FUNCTION_BLOCK TestPublishValue
  VAR
    MQTT : HANDLE_MQTT;
    MQTT_INFO : MQTT_INFO;
    MQTT_IN_OUT : MQTT_IN_OUT;
    testPiublish : ARRAY[0..100] OF MQTTPublish;  (* testPiublish: SD_MQTT.MQTTPublish; *)
    init : BOOL := FALSE;
    sendTest : BOOL;
    TestValue : ARRAY[0..99] OF MQTTValue;
    testtime : ton;
    i : UDINT;
    qos : QoS := 2;
    sub1 : MQTTSubscribe;
    Values : ARRAY[0..99] OF CommonTypesAndFunctions.ALL_TYPES_UNION;
    temp1 : LREAL;
    tmpPointer : CommonTypesAndFunctions.ALL_TYPES_UNION_POINTER;
    MQTTretain : BOOL := TRUE;
    enable : BOOL;
    ERROR_C : DWORD;
    ERROR_T : BYTE;
    ValueTime : TIME := TIME#5s0ms;
  END_VAR

            MQTT_IN_OUT.ClientID :='testCodesys';
MQTT_IN_OUT.COM_CONFIG.MaxPayloadSize :=50000;
MQTT_IN_OUT.COM_CONFIG.MaxTopicLevels := 200;
//testtime(IN:= , PT:= );
testtime(IN:= NOT testtime.Q AND sendTest, PT:= T#100MS);

//testtime(IN:= NOT testtime.Q AND sendTest, PT:= T#10S);
IF NOT init THEN
	init := TRUE;
	tmpPointer.POINTER_TO_LREAL_T := ADR(temp1);
	TestValue[0].Init(
	Topic:= ADR('Haus/Raum1/Tisch/'), 
	ValueName:= ADR('Temperatur'), 
	ValuePointer:= tmpPointer, 
	ValueType:= CommonTypesAndFunctions.VAR_TYPES.LREAL_T, 
	ValueDiff:= 1, 
	MQTT_IN_OUT:= ADR(MQTT_IN_OUT), 
	DecimalPlace:= 2, 
	QoS:= qos, 
	RetainMqtt:= MQTTretain,
	MinTime:=ValueTime);
	sub1.SetMqttInOut(MQTT_IN_OUT:= ADR(MQTT_IN_OUT));

END_IF
TestValue[0]();


MQTT(
	MQTT_INFO:= MQTT_INFO, 
	MQTT_IN_OUT:= MQTT_IN_OUT, 
	ENABLE:= enable, 
	URL:= 'windows-10-pro:1883', 
	TIMEOUT:= T#5S, 
	ERROR_C=> ERROR_C, 
	ERROR_T=> ERROR_T);
          
END_FUNCTION_BLOCK

FUNCTION_BLOCK TestSubscribeOld
  VAR
    MQTT_IN_OUT : MQTT_IN_OUT;
    subscribe : ARRAY[0..20] OF MQTTSubscribe;
    init : BOOL;
    i : INT;
    recived : ARRAY[0..20] OF BOOL;
    CountSplitTopicSizeExceeded : ULINT;
  END_VAR

            IF NOT init THEN
	init := TRUE;
	FOR i := 0 TO 20 DO
		subscribe[i].SetMqttInOut(MQTT_IN_OUT:= ADR(MQTT_IN_OUT));
	END_FOR
END_IF
//MQTT_IN_OUT.OUT.DataRecived := TRUE;
MQTT_IN_OUT.InFree := TRUE;
(*
MQTT_IN_OUT.OUT.MqttTopic := 'r//test';
//GetSplitTopic(in:= MQTT_IN_OUT.OUT.MqttTopic, Target:= ADR(MQTT_IN_OUT.OUT.Topics), CountSplitTopicSizeExceeded:= ADR(CountSplitTopicSizeExceeded));
i:=0;
subscribe[i](
	Subscribe:= TRUE, 
	Topic:= '+//test', 
	QoSSubscribe:= 0, 
	Payload=> , 
	TopicOut=> , 
	SendTimeout=> , 
	SubscribeFail=> , 
	TopicValid=> , 
	Recived=> recived[i]);
MQTT_IN_OUT.OUT.MqttTopic := '/rest/zt';
//GetSplitTopic(in:= MQTT_IN_OUT.OUT.MqttTopic, Target:= ADR(MQTT_IN_OUT.OUT.Topics), CountSplitTopicSizeExceeded:= ADR(CountSplitTopicSizeExceeded));
i:=i+1;
subscribe[i](
	Subscribe:= TRUE, 
	Topic:= '#', 
	QoSSubscribe:= 0, 
	Payload=> , 
	TopicOut=> , 
	SendTimeout=> , 
	SubscribeFail=> , 
	TopicValid=> , 
	Recived=> recived[i]);
MQTT_IN_OUT.OUT.MqttTopic := '566//test/3565/356';
//GetSplitTopic(in:= MQTT_IN_OUT.OUT.MqttTopic, Target:= ADR(MQTT_IN_OUT.OUT.Topics), CountSplitTopicSizeExceeded:= ADR(CountSplitTopicSizeExceeded));
i:=i+1;
subscribe[i](
	Subscribe:= TRUE, 
	Topic:= '+//test/#', 
	QoSSubscribe:= 0, 
	Payload=> , 
	TopicOut=> , 
	SendTimeout=> , 
	SubscribeFail=> , 
	TopicValid=> , 
	Recived=> recived[i]);
MQTT_IN_OUT.OUT.MqttTopic := 'test';
//GetSplitTopic(in:= MQTT_IN_OUT.OUT.MqttTopic, Target:= ADR(MQTT_IN_OUT.OUT.Topics), CountSplitTopicSizeExceeded:= ADR(CountSplitTopicSizeExceeded));
i:=i+1;
subscribe[i](
	Subscribe:= TRUE, 
	Topic:= 'test', 
	QoSSubscribe:= 0, 
	Payload=> , 
	TopicOut=> , 
	SendTimeout=> , 
	SubscribeFail=> , 
	TopicValid=> , 
	Recived=> recived[i]);
MQTT_IN_OUT.OUT.MqttTopic := '/test/';
//GetSplitTopic(in:= MQTT_IN_OUT.OUT.MqttTopic, Target:= ADR(MQTT_IN_OUT.OUT.Topics), CountSplitTopicSizeExceeded:= ADR(CountSplitTopicSizeExceeded));
i:=i+1;
subscribe[i](
	Subscribe:= TRUE, 
	Topic:= 'test/', 
	QoSSubscribe:= 0, 
	Payload=> , 
	TopicOut=> , 
	SendTimeout=> , 
	SubscribeFail=> , 
	TopicValid=> , 
	Recived=> recived[i]);
MQTT_IN_OUT.OUT.MqttTopic := 'test/test1';
//GetSplitTopic(in:= MQTT_IN_OUT.OUT.MqttTopic, Target:= ADR(MQTT_IN_OUT.OUT.Topics), CountSplitTopicSizeExceeded:= ADR(CountSplitTopicSizeExceeded));
i:=i+1;
subscribe[i](
	Subscribe:= TRUE, 
	Topic:= 'test/test1', 
	QoSSubscribe:= 0, 
	Payload=> , 
	TopicOut=> , 
	SendTimeout=> , 
	SubscribeFail=> , 
	TopicValid=> , 
	Recived=> recived[i]);
MQTT_IN_OUT.OUT.MqttTopic := 'a/ret/test';
//GetSplitTopic(in:= MQTT_IN_OUT.OUT.MqttTopic, Target:= ADR(MQTT_IN_OUT.OUT.Topics), CountSplitTopicSizeExceeded:= ADR(CountSplitTopicSizeExceeded));
i:=i+1;
subscribe[i](
	Subscribe:= TRUE, 
	Topic:= 'a/+/test', 
	QoSSubscribe:= 0, 
	Payload=> , 
	TopicOut=> , 
	SendTimeout=> , 
	SubscribeFail=> , 
	TopicValid=> , 
	Recived=> recived[i]);
MQTT_IN_OUT.OUT.MqttTopic := '/test/etwetre/';
//GetSplitTopic(in:= MQTT_IN_OUT.OUT.MqttTopic, Target:= ADR(MQTT_IN_OUT.OUT.Topics), CountSplitTopicSizeExceeded:= ADR(CountSplitTopicSizeExceeded));
i:=i+1;
subscribe[i](
	Subscribe:= TRUE, 
	Topic:= '/test/+',//no match !!!!!
	QoSSubscribe:= 0, 
	Payload=> , 
	TopicOut=> , 
	SendTimeout=> , 
	SubscribeFail=> , 
	TopicValid=> , 
	Recived=> recived[i]);
MQTT_IN_OUT.OUT.MqttTopic := '/test/etwetre';
//GetSplitTopic(in:= MQTT_IN_OUT.OUT.MqttTopic, Target:= ADR(MQTT_IN_OUT.OUT.Topics), CountSplitTopicSizeExceeded:= ADR(CountSplitTopicSizeExceeded));
i:=i+1;
subscribe[i](
	Subscribe:= TRUE, 
	Topic:= '/test/+',//match !!!!!!
	QoSSubscribe:= 0, 
	Payload=> , 
	TopicOut=> , 
	SendTimeout=> , 
	SubscribeFail=> , 
	TopicValid=> , 
	Recived=> recived[i]);
MQTT_IN_OUT.OUT.MqttTopic := '/finance';
//GetSplitTopic(in:= MQTT_IN_OUT.OUT.MqttTopic, Target:= ADR(MQTT_IN_OUT.OUT.Topics), CountSplitTopicSizeExceeded:= ADR(CountSplitTopicSizeExceeded));
i:=i+1;
subscribe[i](
	Subscribe:= TRUE, 
	Topic:= '+/+', //match
	QoSSubscribe:= 0, 
	Payload=> , 
	TopicOut=> , 
	SendTimeout=> , 
	SubscribeFail=> , 
	TopicValid=> , 
	Recived=> recived[i]);
MQTT_IN_OUT.OUT.MqttTopic := '/finance';
//GetSplitTopic(in:= MQTT_IN_OUT.OUT.MqttTopic, Target:= ADR(MQTT_IN_OUT.OUT.Topics), CountSplitTopicSizeExceeded:= ADR(CountSplitTopicSizeExceeded));
i:=i+1;
subscribe[i](
	Subscribe:= TRUE, 
	Topic:= '/+', //match
	QoSSubscribe:= 0, 
	Payload=> , 
	TopicOut=> , 
	SendTimeout=> , 
	SubscribeFail=> , 
	TopicValid=> , 
	Recived=> recived[i]);
MQTT_IN_OUT.OUT.MqttTopic := '/finance';
//GetSplitTopic(in:= MQTT_IN_OUT.OUT.MqttTopic, Target:= ADR(MQTT_IN_OUT.OUT.Topics), CountSplitTopicSizeExceeded:= ADR(CountSplitTopicSizeExceeded));
i:=i+1;
subscribe[i](
	Subscribe:= TRUE, 
	Topic:= '+',//no match 
	QoSSubscribe:= 0, 
	Payload=> , 
	TopicOut=> , 
	SendTimeout=> , 
	SubscribeFail=> , 
	TopicValid=> , 
	Recived=> recived[i]);
MQTT_IN_OUT.OUT.MqttTopic := 'finance/test';
//GetSplitTopic(in:= MQTT_IN_OUT.OUT.MqttTopic, Target:= ADR(MQTT_IN_OUT.OUT.Topics), CountSplitTopicSizeExceeded:= ADR(CountSplitTopicSizeExceeded));
i:=i+1;
subscribe[i](
	Subscribe:= TRUE, 
	Topic:= 'finance/test/',//** 
	QoSSubscribe:= 0, 
	Payload=> , 
	TopicOut=> , 
	SendTimeout=> , 
	SubscribeFail=> , 
	TopicValid=> , 
	Recived=> recived[i]);
MQTT_IN_OUT.OUT.MqttTopic := 'finance/test';
//GetSplitTopic(in:= MQTT_IN_OUT.OUT.MqttTopic, Target:= ADR(MQTT_IN_OUT.OUT.Topics), CountSplitTopicSizeExceeded:= ADR(CountSplitTopicSizeExceeded));
i:=i+1;
subscribe[i](
	Subscribe:= TRUE, 
	Topic:= 'finance/test',//?? 
	QoSSubscribe:= 0, 
	Payload=> , 
	TopicOut=> , 
	SendTimeout=> , 
	SubscribeFail=> , 
	TopicValid=> , 
	Recived=> recived[i]);
MQTT_IN_OUT.OUT.MqttTopic := 'finance/test';
//GetSplitTopic(in:= MQTT_IN_OUT.OUT.MqttTopic, Target:= ADR(MQTT_IN_OUT.OUT.Topics), CountSplitTopicSizeExceeded:= ADR(CountSplitTopicSizeExceeded));
i:=i+1;
subscribe[i](
	Subscribe:= TRUE, 
	Topic:= 'finance/test/+',//?? 
	QoSSubscribe:= 0, 
	Payload=> , 
	TopicOut=> , 
	SendTimeout=> , 
	SubscribeFail=> , 
	TopicValid=> , 
	Recived=> recived[i]);

MQTT_IN_OUT.OUT.MqttTopic := 'finance';
//GetSplitTopic(in:= MQTT_IN_OUT.OUT.MqttTopic, Target:= ADR(MQTT_IN_OUT.OUT.Topics), CountSplitTopicSizeExceeded:= ADR(CountSplitTopicSizeExceeded));
i:=i+1;
subscribe[i](
	Subscribe:= TRUE, 
	Topic:= 'finance/#',//?match
	QoSSubscribe:= 0, 
	Payload=> , 
	TopicOut=> , 
	SendTimeout=> , 
	SubscribeFail=> , 
	TopicValid=> , 
	Recived=> recived[i]);
MQTT_IN_OUT.OUT.MqttTopic := 'finance/';
//GetSplitTopic(in:= MQTT_IN_OUT.OUT.MqttTopic, Target:= ADR(MQTT_IN_OUT.OUT.Topics), CountSplitTopicSizeExceeded:= ADR(CountSplitTopicSizeExceeded));
i:=i+1;
subscribe[i](
	Subscribe:= TRUE, 
	Topic:= 'finance/#',// match 
	QoSSubscribe:= 0, 
	Payload=> , 
	TopicOut=> , 
	SendTimeout=> , 
	SubscribeFail=> , 
	TopicValid=> , 
	Recived=> recived[i]);
MQTT_IN_OUT.OUT.MqttTopic := 'test/ff';
//GetSplitTopic(in:= MQTT_IN_OUT.OUT.MqttTopic, Target:= ADR(MQTT_IN_OUT.OUT.Topics), CountSplitTopicSizeExceeded:= ADR(CountSplitTopicSizeExceeded));
i:=i+1;
subscribe[i](
	Subscribe:= TRUE, 
	Topic:= 'test/ff/+',//no match 
	QoSSubscribe:= 0, 
	Payload=> , 
	TopicOut=> , 
	SendTimeout=> , 
	SubscribeFail=> , 
	TopicValid=> , 
	Recived=> recived[i]);
MQTT_IN_OUT.OUT.MqttTopic := 'test/ff';
//GetSplitTopic(in:= MQTT_IN_OUT.OUT.MqttTopic, Target:= ADR(MQTT_IN_OUT.OUT.Topics), CountSplitTopicSizeExceeded:= ADR(CountSplitTopicSizeExceeded));
i:=i+1;
subscribe[i](
	Subscribe:= TRUE, 
	Topic:= 'test/ff/#',//match 
	QoSSubscribe:= 0, 
	Payload=> , 
	TopicOut=> , 
	SendTimeout=> , 
	SubscribeFail=> , 
	TopicValid=> , 
	Recived=> recived[i]);
*)
          
END_FUNCTION_BLOCK

FUNCTION_BLOCK TestTopicMatch
  VAR
    t1 : HandleSplitTopic;
    t2 : HandleSplitTopic;
    match : TOPIC_MATCH;
    pts : ARRAY[0..20] OF POINTER TO STRING;
    sp : POINTER TO SPLIT_TOPIC;
    COM_CONFIG : COM_CONFIG;
    dynMemUsage : UDINT;
  END_VAR

            t1.FullInit(TopicsLevelInit:= 40, SplitElementSizeInit:= 5000, dynMemUsageInit:= ADR(dynMemUsage));
t2.FullInit(TopicsLevelInit:= 40, SplitElementSizeInit:= 5000, dynMemUsageInit:= ADR(dynMemUsage));


t1.NewTopic(in:=ADR('/+/test/#'),test:= TRUE, SizeOfString:= 0);
	sp := t1.GetSplitTopic();
	pts[0] := sp^.Topics[0];
	pts[1] := sp^.Topics[1];
	pts[2] := sp^.Topics[2];
	pts[3] := sp^.Topics[3];
	pts[4] := sp^.Topics[4];
	pts[5] := sp^.Topics[5];
	pts[6] := sp^.Topics[6];
	pts[7] := sp^.Topics[7];
	pts[8] := sp^.Topics[8];
t2.NewTopic(in:=ADR('/rtt/test/tr'),test:= FALSE, SizeOfString:= 0);
	sp := t2.GetSplitTopic();
	pts[10] := sp^.Topics[0];
	pts[11] := sp^.Topics[1];
	pts[12] := sp^.Topics[2];
	pts[13] := sp^.Topics[3];
	pts[14] := sp^.Topics[4];
	pts[15] := sp^.Topics[5];
	pts[16] := sp^.Topics[6];
	pts[17] := sp^.Topics[7];
	pts[18] := sp^.Topics[8];
match := t1.CheckTopicMatchToMe(with:= t2.GetSplitTopic());


//test from MQTT doku
t1.NewTopic(in:=ADR('sport/tennis/+'),test:= TRUE, SizeOfString:= 0);
t2.NewTopic(in:=ADR('sport/tennis/player1'),test:= FALSE, SizeOfString:= 0);
match := t1.CheckTopicMatchToMe(with:= t2.GetSplitTopic()); //match
t2.NewTopic(in:=ADR('sport/tennis/player2'),test:= FALSE, SizeOfString:= 0);
match := t1.CheckTopicMatchToMe(with:= t2.GetSplitTopic());//match
t2.NewTopic(in:=ADR('sport/tennis/player1/ranking'),test:= FALSE, SizeOfString:= 0);
match := t1.CheckTopicMatchToMe(with:= t2.GetSplitTopic());//no match


t1.NewTopic(in:=ADR('sport/+'),test:= TRUE, SizeOfString:= 0);
t2.NewTopic(in:=ADR('sport'),test:= FALSE, SizeOfString:= 0);
match := t1.CheckTopicMatchToMe(with:= t2.GetSplitTopic()); //no match

t2.NewTopic(in:=ADR('sport/'),test:= FALSE, SizeOfString:= 0);
match := t1.CheckTopicMatchToMe(with:= t2.GetSplitTopic()); //match

t1.NewTopic(in:=ADR('+/+'),test:= TRUE, SizeOfString:= 0);
t2.NewTopic(in:=ADR('/finance'),test:= FALSE, SizeOfString:= 0);
match := t1.CheckTopicMatchToMe(with:= t2.GetSplitTopic()); //match

t1.NewTopic(in:=ADR('/+'),test:= TRUE, SizeOfString:= 0);
match := t1.CheckTopicMatchToMe(with:= t2.GetSplitTopic()); //match

t1.NewTopic(in:=ADR('+'),test:= TRUE, SizeOfString:= 0);
match := t1.CheckTopicMatchToMe(with:= t2.GetSplitTopic()); //no match
//just for breakpoint
t1.NewTopic(in:=ADR('+/+'),test:= TRUE, SizeOfString:= 0);



          
END_FUNCTION_BLOCK
